PROGRAM MAIN
VAR
END_VAR

Shutdown();

END_PROGRAM

(* stored: Version 1.1.0.1, ProductVersion 3.1.4022.3
   POU MAIN: Id {8543b332-675f-49bb-9ec1-b605778f4250}, SpecialFunc None *)
